FUNCTION_BLOCK CL_CGSSystemBase EXTENDS CL_MasterRootClass
VAR
  //INTERNAL VAR
  _stSystemStatus_ARR   : ST_SystemStatus_ARR;
  bInitSysBase          : BOOL := FALSE;
END_VAR

//State machine history
IF bInitSysBase THEN 
  //Manage Mode machine
  IF _stSystemStatus_ARR[MRIrrLine].nRequestModeMachine <> nModeMachine AND _stSystemStatus_ARR[MRIrrLine].nStateMachine = E_StateMachine.cStopped THEN
    _stSystemStatus_ARR[MRIrrLine].nModeMachine := _stSystemStatus_ARR[MRIrrLine].nRequestModeMachine;
  END_IF  
END_IF

METHOD PUBLIC InitSystemBase : BOOL
VAR_INPUT
  //nIrrLine             : UINT := 0;
  //nIrrLineFixedID      : UINT := 0;
  IrrLine              : ST_LineReference;
  stSystemStatus_ARR   : ST_SystemStatus_ARR;
END_VAR
InitSystemBase := FALSE;
IF __ISVALIDREF(stSystemStatus_ARR) AND NOT bInitSysBase 
   AND IrrLine.nThis >= 0 AND IrrLine.nThis <= C.uiNumIrrLinesForHMI_C
   AND IrrLine.nFixedID >= 0 AND IrrLine.nThis <= C.uiNumIrrLinesInGreenhouse_C THEN
    _stSystemStatus_ARR REF= stSystemStatus_ARR;
    MRLineRef := IrrLine;
    InitSystemBase := bInitSysBase := TRUE;
END_IF
END_METHOD

PROPERTY PUBLIC nModeMachine : E_ModeMachine
GET
IF bInitSysBase THEN 
  nModeMachine := _stSystemStatus_ARR[MRIrrLine].nModeMachine;
ELSE
  nModeMachine := E_ModeMachine.Startup;
END_IF
END_GET
SET
IF bInitSysBase THEN 
  _stSystemStatus_ARR[MRIrrLine].nModeMachine := nModeMachine;
ELSE
  _stSystemStatus_ARR[MRIrrLine].nModeMachine := E_ModeMachine.Startup;
END_IF
END_SET
END_PROPERTY

PROPERTY PUBLIC nReqModeMachine : E_ModeMachine
GET
IF bInitSysBase THEN 
  nReqModeMachine := _stSystemStatus_ARR[MRIrrLine].nRequestModeMachine;
ELSE
  nReqModeMachine := E_ModeMachine.Startup;
END_IF
END_GET
SET
IF bInitSysBase THEN 
  _stSystemStatus_ARR[MRIrrLine].nRequestModeMachine := nReqModeMachine;
ELSE
 _stSystemStatus_ARR[MRIrrLine].nRequestModeMachine := E_ModeMachine.Startup;
END_IF
END_SET
END_PROPERTY

PROPERTY PUBLIC nStateMachine : E_StateMachine
GET
IF bInitSysBase THEN 
  nStateMachine := _stSystemStatus_ARR[MRIrrLine].nStateMachine;
ELSE
  nStateMachine := E_StateMachine.cIdle;
END_IF
END_GET
SET
IF bInitSysBase THEN 
  _stSystemStatus_ARR[MRIrrLine].nStateMachine := nStateMachine;
ELSE
  _stSystemStatus_ARR[MRIrrLine].nStateMachine := E_StateMachine.cIdle;;
END_IF
END_SET
END_PROPERTY

METHOD PUBLIC ReqModeMachine : BOOL
VAR_INPUT
  nModeMachine   : E_ModeMachine;;
END_VAR
IF bInitSysBase THEN 
  _stSystemStatus_ARR[MRIrrLine].nRequestModeMachine := nModeMachine;
END_IF
END_METHOD

END_FUNCTION_BLOCK

(* stored: Version 1.1.0.1, ProductVersion 3.1.4024.12
   POU CL_CGSSystemBase: Id {649a3c98-cef9-49ef-abcc-66e50a4447d0}, SpecialFunc None
   Method InitSystemBase: Id {dc707108-b7f1-4495-812f-276911c5d8f9}
   Property nModeMachine: Id {6ccbbe11-206f-4ece-886c-b3c198b618bd}
   Get Get: Id {e5d8187a-c430-43e9-aea1-e8db6ec3bf3e}
   Set Set: Id {274c2497-a6f8-4743-82d8-aaeef5ae1292}
   Property nReqModeMachine: Id {7dc10879-510f-4ea6-b155-6b3b01fd4ecb}
   Get Get: Id {d0b08a63-2027-4daf-9fa0-a6556310478c}
   Set Set: Id {be73520c-eec3-4e60-bf9b-d9cbbb89c345}
   Property nStateMachine: Id {b22ca0d4-44a4-40c1-a42d-9361fd4d5108}
   Get Get: Id {5ff9b98b-39b3-4b78-a3b5-7b9e8ea604ac}
   Set Set: Id {a4bd60e8-afdc-4af0-a573-39811e224709}
   Method ReqModeMachine: Id {a96c1e55-f3b4-4370-a009-07d0ab47c4fc} *)
